(* PLC project  *)

CONFIGURATION EL2809
END_CONFIGURATION
